// TIA Portal V18 export
TYPE "UDT_WeatherCompCurve"
// stored: IsFailsafeCompliant false
   STRUCT
      rEffectiveRoomSetPoint : Array[0..2] of Real;
      rHeatingCurveLevel : Array[0..2] of Real;
      rHeatingCurveSlope : Array[0..2] of Real;
      rSetpointTemp : Array[0..2] of Real;
      rOATforHeatingCurves : Array[0..2] of Real;
   END_STRUCT;
   // rEffectiveRoomSetPoint[0] := 20.0;
   // rEffectiveRoomSetPoint[1] := 21.0;
   // rEffectiveRoomSetPoint[2] := 22.0;
   // rHeatingCurveLevel[1] := 1.0;
   // rHeatingCurveLevel[2] := 2.0;
   // rHeatingCurveSlope[0] := 2.0;
   // rHeatingCurveSlope[1] := 2.1;
   // rHeatingCurveSlope[2] := 2.2;
   // rSetpointTemp[0] := 50.0;
   // rSetpointTemp[1] := 51.0;
   // rSetpointTemp[2] := 52.0;
END_TYPE
